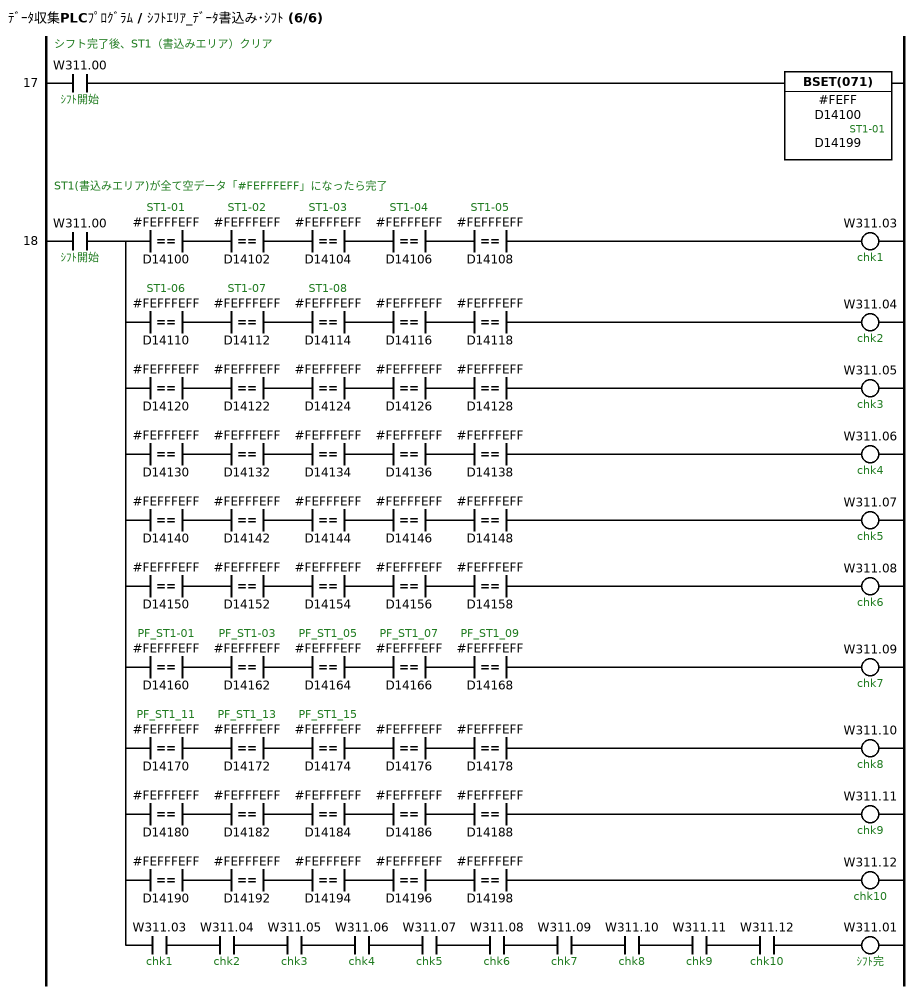
; [picture p24: ﾃﾞｰﾀ収集PLCﾌﾟﾛｸﾞﾗﾑ / ｼﾌﾄｴﾘｱ_ﾃﾞｰﾀ書込み･ｼﾌﾄ, rungs 17-18]
; rung 17: シフト完了後、ST1（書込みエリア）クリア
LD W311.00  ; ｼﾌﾄ開始
BSET(071) #FEFF D14100 D14199  ; ST1-01
; rung 18: ST1(書込みエリア)が全て空データ「#FEFFFEFF」になったら完了
LD W311.00  ; ｼﾌﾄ開始
OUT TR0
AND=L(301) #FEFFFEFF D14100  ; ST1-01
AND=L(301) #FEFFFEFF D14102  ; ST1-02
AND=L(301) #FEFFFEFF D14104  ; ST1-03
AND=L(301) #FEFFFEFF D14106  ; ST1-04
AND=L(301) #FEFFFEFF D14108  ; ST1-05
OUT W311.03  ; chk1
LD TR0
AND=L(301) #FEFFFEFF D14110  ; ST1-06
AND=L(301) #FEFFFEFF D14112  ; ST1-07
AND=L(301) #FEFFFEFF D14114  ; ST1-08
AND=L(301) #FEFFFEFF D14116
AND=L(301) #FEFFFEFF D14118
OUT W311.04  ; chk2
LD TR0
AND=L(301) #FEFFFEFF D14120
AND=L(301) #FEFFFEFF D14122
AND=L(301) #FEFFFEFF D14124
AND=L(301) #FEFFFEFF D14126
AND=L(301) #FEFFFEFF D14128
OUT W311.05  ; chk3
LD TR0
AND=L(301) #FEFFFEFF D14130
AND=L(301) #FEFFFEFF D14132
AND=L(301) #FEFFFEFF D14134
AND=L(301) #FEFFFEFF D14136
AND=L(301) #FEFFFEFF D14138
OUT W311.06  ; chk4
LD TR0
AND=L(301) #FEFFFEFF D14140
AND=L(301) #FEFFFEFF D14142
AND=L(301) #FEFFFEFF D14144
AND=L(301) #FEFFFEFF D14146
AND=L(301) #FEFFFEFF D14148
OUT W311.07  ; chk5
LD TR0
AND=L(301) #FEFFFEFF D14150
AND=L(301) #FEFFFEFF D14152
AND=L(301) #FEFFFEFF D14154
AND=L(301) #FEFFFEFF D14156
AND=L(301) #FEFFFEFF D14158
OUT W311.08  ; chk6
LD TR0
AND=L(301) #FEFFFEFF D14160  ; PF_ST1-01
AND=L(301) #FEFFFEFF D14162  ; PF_ST1-03
AND=L(301) #FEFFFEFF D14164  ; PF_ST1_05
AND=L(301) #FEFFFEFF D14166  ; PF_ST1_07
AND=L(301) #FEFFFEFF D14168  ; PF_ST1_09
OUT W311.09  ; chk7
LD TR0
AND=L(301) #FEFFFEFF D14170  ; PF_ST1_11
AND=L(301) #FEFFFEFF D14172  ; PF_ST1_13
AND=L(301) #FEFFFEFF D14174  ; PF_ST1_15
AND=L(301) #FEFFFEFF D14176
AND=L(301) #FEFFFEFF D14178
OUT W311.10  ; chk8
LD TR0
AND=L(301) #FEFFFEFF D14180
AND=L(301) #FEFFFEFF D14182
AND=L(301) #FEFFFEFF D14184
AND=L(301) #FEFFFEFF D14186
AND=L(301) #FEFFFEFF D14188
OUT W311.11  ; chk9
LD TR0
AND=L(301) #FEFFFEFF D14190
AND=L(301) #FEFFFEFF D14192
AND=L(301) #FEFFFEFF D14194
AND=L(301) #FEFFFEFF D14196
AND=L(301) #FEFFFEFF D14198
OUT W311.12  ; chk10
LD TR0
AND W311.03  ; chk1
AND W311.04  ; chk2
AND W311.05  ; chk3
AND W311.06  ; chk4
AND W311.07  ; chk5
AND W311.08  ; chk6
AND W311.09  ; chk7
AND W311.10  ; chk8
AND W311.11  ; chk9
AND W311.12  ; chk10
OUT W311.01  ; ｼﾌﾄ完

### Section ｼﾌﾄｴﾘｱ_ﾃﾞｰﾀ読出し

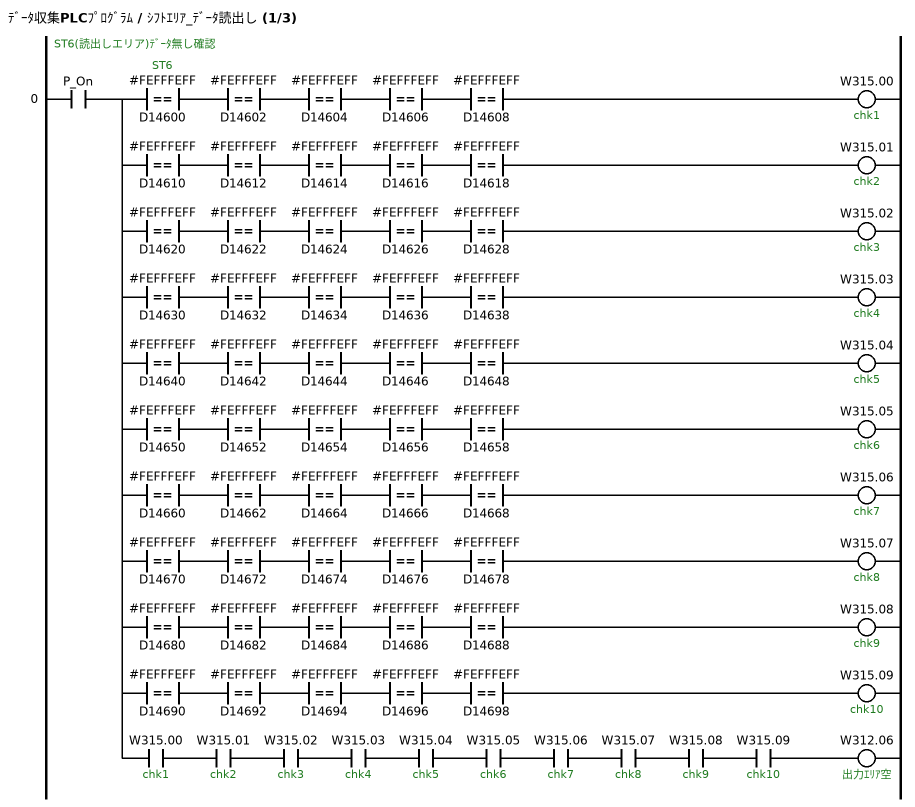
; rung 0: ST6(読出しエリア)ﾃﾞｰﾀ無し確認
LD P_On
OUT TR0
AND=L(301) #FEFFFEFF D14600  ; ST6
AND=L(301) #FEFFFEFF D14602
AND=L(301) #FEFFFEFF D14604
AND=L(301) #FEFFFEFF D14606
AND=L(301) #FEFFFEFF D14608
OUT W315.00  ; chk1
LD TR0
AND=L(301) #FEFFFEFF D14610
AND=L(301) #FEFFFEFF D14612
AND=L(301) #FEFFFEFF D14614
AND=L(301) #FEFFFEFF D14616
AND=L(301) #FEFFFEFF D14618
OUT W315.01  ; chk2
LD TR0
AND=L(301) #FEFFFEFF D14620
AND=L(301) #FEFFFEFF D14622
AND=L(301) #FEFFFEFF D14624
AND=L(301) #FEFFFEFF D14626
AND=L(301) #FEFFFEFF D14628
OUT W315.02  ; chk3
LD TR0
AND=L(301) #FEFFFEFF D14630
AND=L(301) #FEFFFEFF D14632
AND=L(301) #FEFFFEFF D14634
AND=L(301) #FEFFFEFF D14636
AND=L(301) #FEFFFEFF D14638
OUT W315.03  ; chk4
LD TR0
AND=L(301) #FEFFFEFF D14640
AND=L(301) #FEFFFEFF D14642
AND=L(301) #FEFFFEFF D14644
AND=L(301) #FEFFFEFF D14646
AND=L(301) #FEFFFEFF D14648
OUT W315.04  ; chk5
LD TR0
AND=L(301) #FEFFFEFF D14650
AND=L(301) #FEFFFEFF D14652
AND=L(301) #FEFFFEFF D14654
AND=L(301) #FEFFFEFF D14656
AND=L(301) #FEFFFEFF D14658
OUT W315.05  ; chk6
LD TR0
AND=L(301) #FEFFFEFF D14660
AND=L(301) #FEFFFEFF D14662
AND=L(301) #FEFFFEFF D14664
AND=L(301) #FEFFFEFF D14666
AND=L(301) #FEFFFEFF D14668
OUT W315.06  ; chk7
LD TR0
AND=L(301) #FEFFFEFF D14670
AND=L(301) #FEFFFEFF D14672
AND=L(301) #FEFFFEFF D14674
AND=L(301) #FEFFFEFF D14676
AND=L(301) #FEFFFEFF D14678
OUT W315.07  ; chk8
LD TR0
AND=L(301) #FEFFFEFF D14680
AND=L(301) #FEFFFEFF D14682
AND=L(301) #FEFFFEFF D14684
AND=L(301) #FEFFFEFF D14686
AND=L(301) #FEFFFEFF D14688
OUT W315.08  ; chk9
LD TR0
AND=L(301) #FEFFFEFF D14690
AND=L(301) #FEFFFEFF D14692
AND=L(301) #FEFFFEFF D14694
AND=L(301) #FEFFFEFF D14696
AND=L(301) #FEFFFEFF D14698
OUT W315.09  ; chk10
LD TR0
AND W315.00  ; chk1
AND W315.01  ; chk2
AND W315.02  ; chk3
AND W315.03  ; chk4
AND W315.04  ; chk5
AND W315.05  ; chk6
AND W315.06  ; chk7
AND W315.07  ; chk8
AND W315.08  ; chk9
AND W315.09  ; chk10
OUT W312.06  ; 出力ｴﾘｱ空

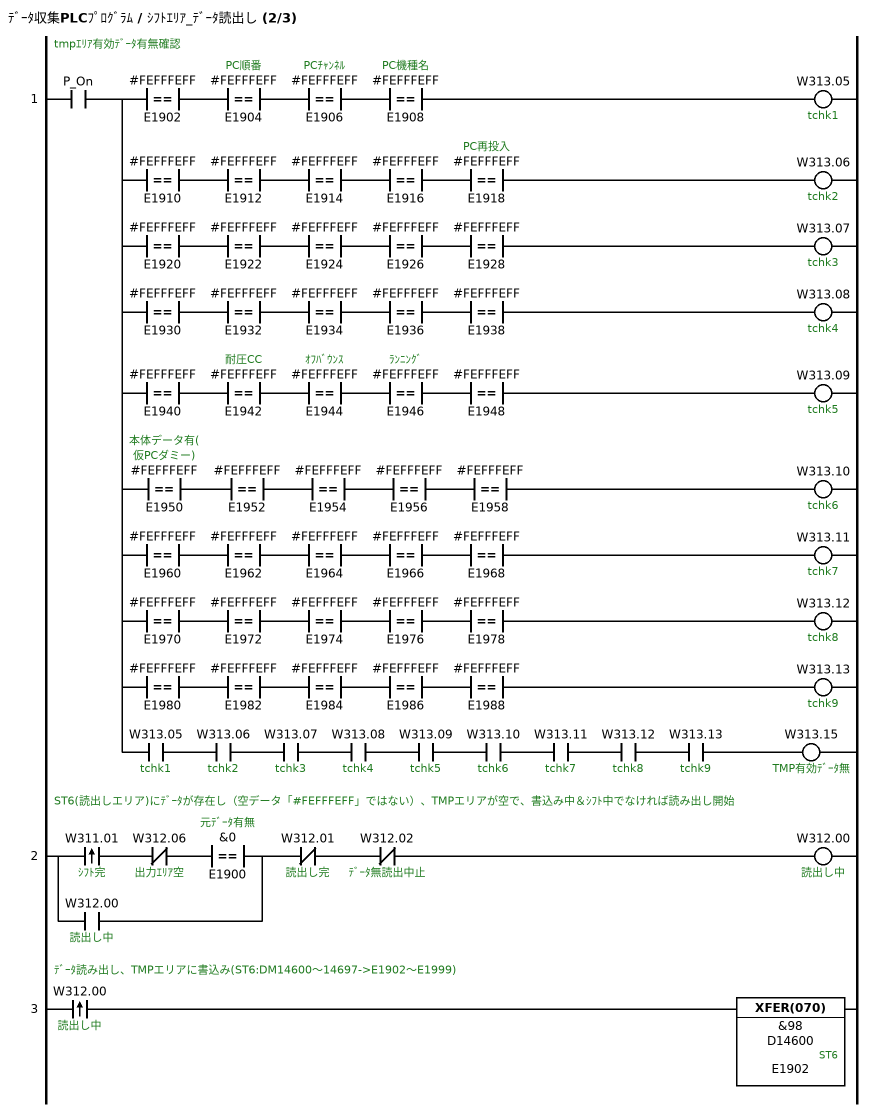
; rung 1: tmpｴﾘｱ有効ﾃﾞｰﾀ有無確認
LD P_On
OUT TR0
AND=L(301) #FEFFFEFF E1902
AND=L(301) #FEFFFEFF E1904  ; PC順番
AND=L(301) #FEFFFEFF E1906  ; PCﾁｬﾝﾈﾙ
AND=L(301) #FEFFFEFF E1908  ; PC機種名
OUT W313.05  ; tchk1
LD TR0
AND=L(301) #FEFFFEFF E1910
AND=L(301) #FEFFFEFF E1912
AND=L(301) #FEFFFEFF E1914
AND=L(301) #FEFFFEFF E1916
AND=L(301) #FEFFFEFF E1918  ; PC再投入
OUT W313.06  ; tchk2
LD TR0
AND=L(301) #FEFFFEFF E1920
AND=L(301) #FEFFFEFF E1922
AND=L(301) #FEFFFEFF E1924
AND=L(301) #FEFFFEFF E1926
AND=L(301) #FEFFFEFF E1928
OUT W313.07  ; tchk3
LD TR0
AND=L(301) #FEFFFEFF E1930
AND=L(301) #FEFFFEFF E1932
AND=L(301) #FEFFFEFF E1934
AND=L(301) #FEFFFEFF E1936
AND=L(301) #FEFFFEFF E1938
OUT W313.08  ; tchk4
LD TR0
AND=L(301) #FEFFFEFF E1940
AND=L(301) #FEFFFEFF E1942  ; 耐圧CC
AND=L(301) #FEFFFEFF E1944  ; ｵﾌﾊﾞｳﾝｽ
AND=L(301) #FEFFFEFF E1946  ; ﾗﾝﾆﾝｸﾞ
AND=L(301) #FEFFFEFF E1948
OUT W313.09  ; tchk5
LD TR0
AND=L(301) #FEFFFEFF E1950  ; 本体データ有(仮PCダミー)
AND=L(301) #FEFFFEFF E1952
AND=L(301) #FEFFFEFF E1954
AND=L(301) #FEFFFEFF E1956
AND=L(301) #FEFFFEFF E1958
OUT W313.10  ; tchk6
LD TR0
AND=L(301) #FEFFFEFF E1960
AND=L(301) #FEFFFEFF E1962
AND=L(301) #FEFFFEFF E1964
AND=L(301) #FEFFFEFF E1966
AND=L(301) #FEFFFEFF E1968
OUT W313.11  ; tchk7
LD TR0
AND=L(301) #FEFFFEFF E1970
AND=L(301) #FEFFFEFF E1972
AND=L(301) #FEFFFEFF E1974
AND=L(301) #FEFFFEFF E1976
AND=L(301) #FEFFFEFF E1978
OUT W313.12  ; tchk8
LD TR0
AND=L(301) #FEFFFEFF E1980
AND=L(301) #FEFFFEFF E1982
AND=L(301) #FEFFFEFF E1984
AND=L(301) #FEFFFEFF E1986
AND=L(301) #FEFFFEFF E1988
OUT W313.13  ; tchk9
LD TR0
AND W313.05  ; tchk1
AND W313.06  ; tchk2
AND W313.07  ; tchk3
AND W313.08  ; tchk4
AND W313.09  ; tchk5
AND W313.10  ; tchk6
AND W313.11  ; tchk7
AND W313.12  ; tchk8
AND W313.13  ; tchk9
OUT W313.15  ; TMP有効ﾃﾞｰﾀ無
; rung 2: ST6(読出しエリア)にﾃﾞｰﾀが存在し（空データ「#FEFFFEFF」ではない）、TMPエリアが空で、書込み中＆ｼﾌﾄ中でなければ読み出し開始
@LD W311.01  ; ｼﾌﾄ完
ANDNOT W312.06  ; 出力ｴﾘｱ空
AND=(300) &0 E1900  ; 元ﾃﾞｰﾀ有無
OR W312.00  ; 読出し中
ANDNOT W312.01  ; 読出し完
ANDNOT W312.02  ; ﾃﾞｰﾀ無読出中止
OUT W312.00  ; 読出し中
; rung 3: ﾃﾞｰﾀ読み出し、TMPエリアに書込み(ST6:DM14600～14697->E1902～E1999)
@LD W312.00  ; 読出し中
XFER(070) &98 D14600 E1902  ; ST6

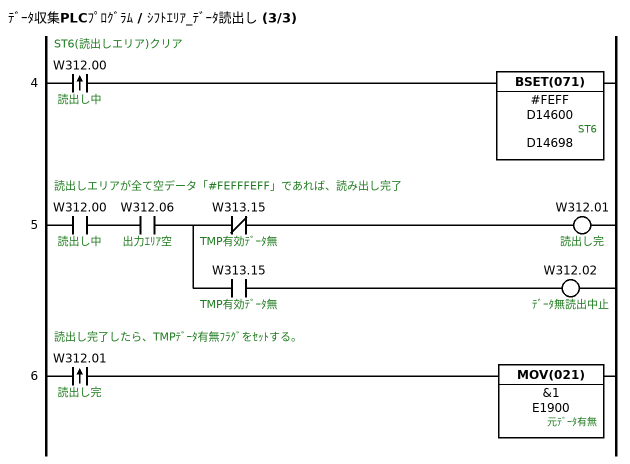
; rung 4: ST6(読出しエリア)クリア
@LD W312.00  ; 読出し中
BSET(071) #FEFF D14600 D14698  ; ST6
; rung 5: 読出しエリアが全て空データ「#FEFFFEFF」であれば、読み出し完了
LD W312.00  ; 読出し中
AND W312.06  ; 出力ｴﾘｱ空
OUT TR0
ANDNOT W313.15  ; TMP有効ﾃﾞｰﾀ無
OUT W312.01  ; 読出し完
LD TR0
AND W313.15  ; TMP有効ﾃﾞｰﾀ無
OUT W312.02  ; ﾃﾞｰﾀ無読出中止
; rung 6: 読出し完了したら、TMPﾃﾞｰﾀ有無ﾌﾗｸﾞをｾｯﾄする。
@LD W312.01  ; 読出し完
MOV(021) &1 E1900  ; 元ﾃﾞｰﾀ有無

### Section ｼﾌﾄｴﾘｱ_ﾃﾞｰﾀｸﾘｱ

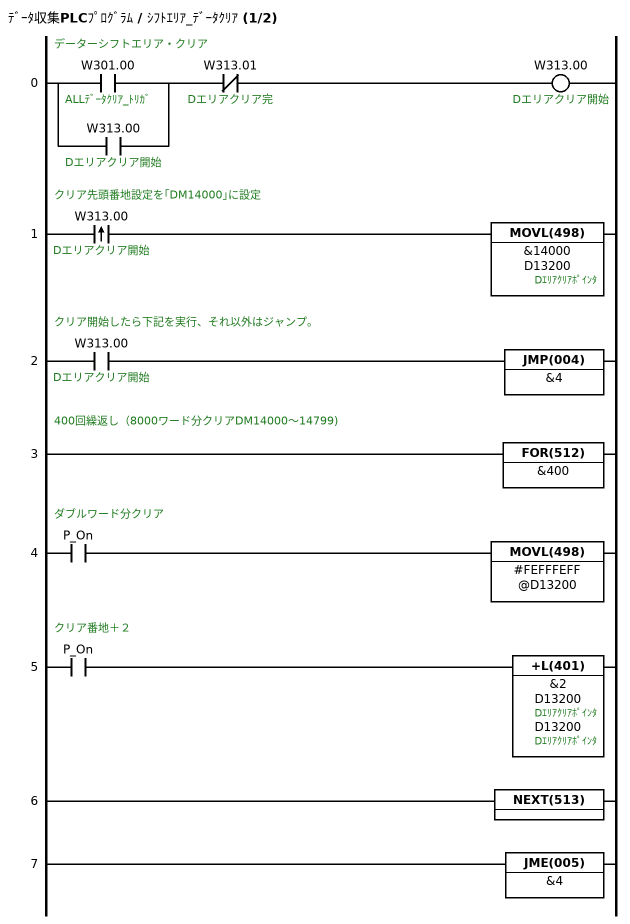
; rung 0: データーシフトエリア・クリア
LD W301.00  ; ALLﾃﾞｰﾀｸﾘｱ_ﾄﾘｶﾞ
OR W313.00  ; Dエリアクリア開始
ANDNOT W313.01  ; Dエリアクリア完
OUT W313.00  ; Dエリアクリア開始
; rung 1: クリア先頭番地設定を｢DM14000｣に設定
@LD W313.00  ; Dエリアクリア開始
MOVL(498) &14000 D13200  ; Dｴﾘｱｸﾘｱﾎﾟｲﾝﾀ
; rung 2: クリア開始したら下記を実行、それ以外はジャンプ。
LD W313.00  ; Dエリアクリア開始
JMP(004) &4
; rung 3: 400回繰返し（8000ワード分クリアDM14000～14799)
FOR(512) &400
; rung 4: ダブルワード分クリア
LD P_On
MOVL(498) #FEFFFEFF @D13200
; rung 5: クリア番地＋２
LD P_On
+L(401) &2 D13200 D13200  ; Dｴﾘｱｸﾘｱﾎﾟｲﾝﾀ
; rung 6
NEXT(513)
; rung 7
JME(005) &4

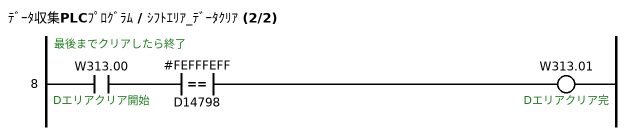
; rung 8: 最後までクリアしたら終了
LD W313.00  ; Dエリアクリア開始
AND=L(301) #FEFFFEFF D14798
OUT W313.01  ; Dエリアクリア完

### Section ｽﾀｯｸｴﾘｱ_ﾃﾞｰﾀ書込み

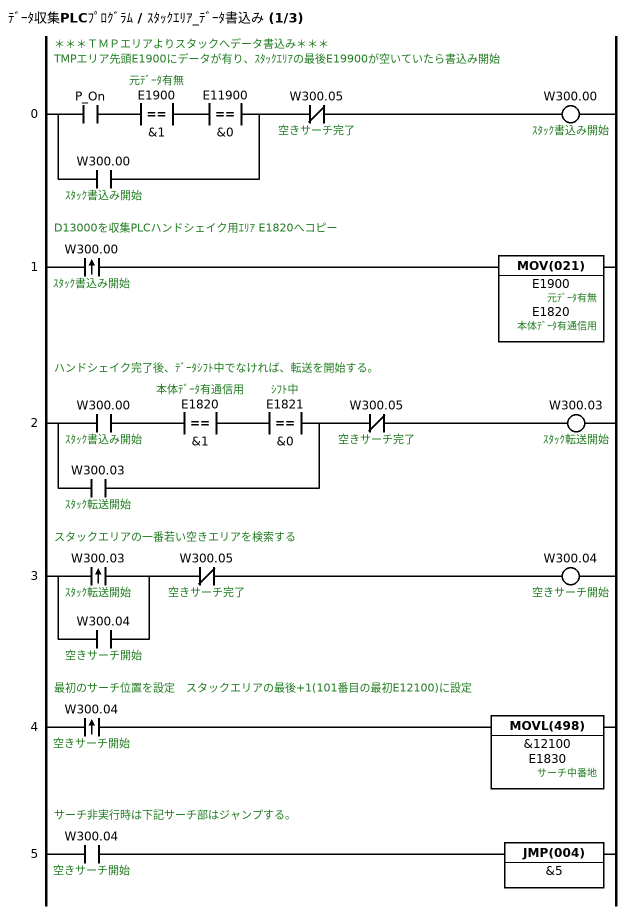
; rung 0: ＊＊＊ＴＭＰエリアよりスタックへデータ書込み＊＊＊ / TMPエリア先頭E1900にデータが有り、ｽﾀｯｸｴﾘｱの最後E19900が空いていたら書込み開始
LD P_On
AND=(300) E1900 &1  ; 元ﾃﾞｰﾀ有無
AND=(300) E11900 &0
OR W300.00  ; ｽﾀｯｸ書込み開始
ANDNOT W300.05  ; 空きサーチ完了
OUT W300.00  ; ｽﾀｯｸ書込み開始
; rung 1: D13000を収集PLCハンドシェイク用ｴﾘｱ E1820へコピー
@LD W300.00  ; ｽﾀｯｸ書込み開始
MOV(021) E1900 E1820  ; 元ﾃﾞｰﾀ有無, 本体ﾃﾞｰﾀ有通信用
; rung 2: ハンドシェイク完了後、ﾃﾞｰﾀｼﾌﾄ中でなければ、転送を開始する。
LD W300.00  ; ｽﾀｯｸ書込み開始
AND=(300) E1820 &1  ; 本体ﾃﾞｰﾀ有通信用
AND=(300) E1821 &0  ; ｼﾌﾄ中
OR W300.03  ; ｽﾀｯｸ転送開始
ANDNOT W300.05  ; 空きサーチ完了
OUT W300.03  ; ｽﾀｯｸ転送開始
; rung 3: スタックエリアの一番若い空きエリアを検索する
@LD W300.03  ; ｽﾀｯｸ転送開始
OR W300.04  ; 空きサーチ開始
ANDNOT W300.05  ; 空きサーチ完了
OUT W300.04  ; 空きサーチ開始
; rung 4: 最初のサーチ位置を設定　スタックエリアの最後+1(101番目の最初E12100)に設定
@LD W300.04  ; 空きサーチ開始
MOVL(498) &12100 E1830  ; サーチ中番地
; rung 5: サーチ非実行時は下記サーチ部はジャンプする。
LD W300.04  ; 空きサーチ開始
JMP(004) &5

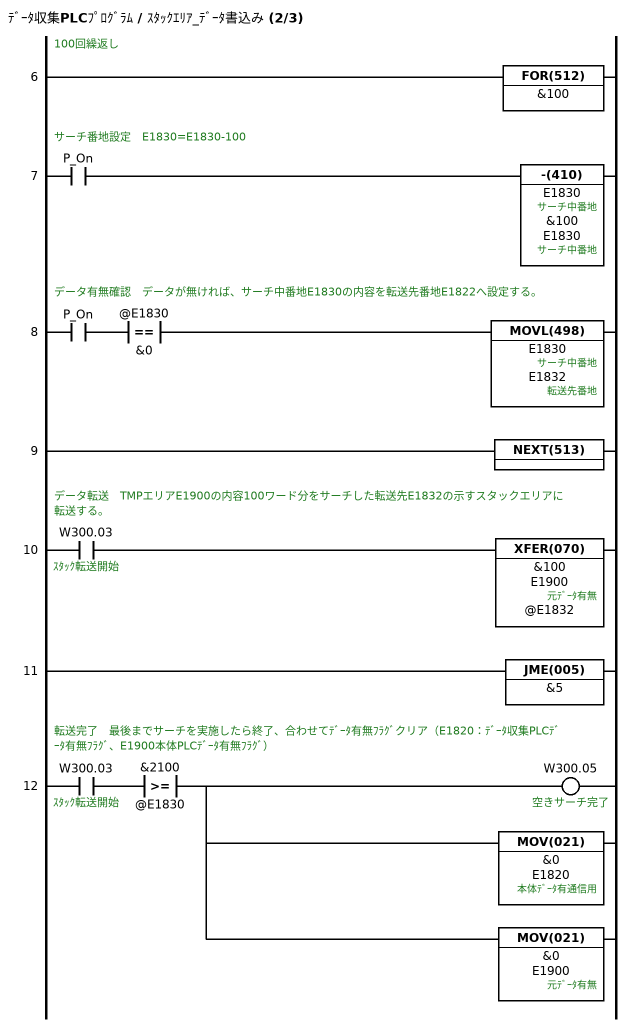
; rung 6: 100回繰返し
FOR(512) &100
; rung 7: サーチ番地設定　E1830=E1830-100
LD P_On
-(410) E1830 &100 E1830  ; サーチ中番地
; rung 8: データ有無確認　データが無ければ、サーチ中番地E1830の内容を転送先番地E1822へ設定する。
LD P_On
AND=(300) @E1830 &0
MOVL(498) E1830 E1832  ; サーチ中番地, 転送先番地
; rung 9
NEXT(513)
; rung 10: データ転送　TMPエリアE1900の内容100ワード分をサーチした転送先E1832の示すスタックエリアに転送する。
LD W300.03  ; ｽﾀｯｸ転送開始
XFER(070) &100 E1900 @E1832  ; 元ﾃﾞｰﾀ有無
; rung 11
JME(005) &5
; rung 12: 転送完了　最後までサーチを実施したら終了、合わせてﾃﾞｰﾀ有無ﾌﾗｸﾞクリア（E1820：ﾃﾞｰﾀ収集PLCﾃﾞｰﾀ有無ﾌﾗｸﾞ、E1900本体PLCﾃﾞｰﾀ有無ﾌﾗｸﾞ）
LD W300.03  ; ｽﾀｯｸ転送開始
AND>=(325) &2100 @E1830
OUT W300.05  ; 空きサーチ完了
MOV(021) &0 E1820  ; 本体ﾃﾞｰﾀ有通信用
MOV(021) &0 E1900  ; 元ﾃﾞｰﾀ有無

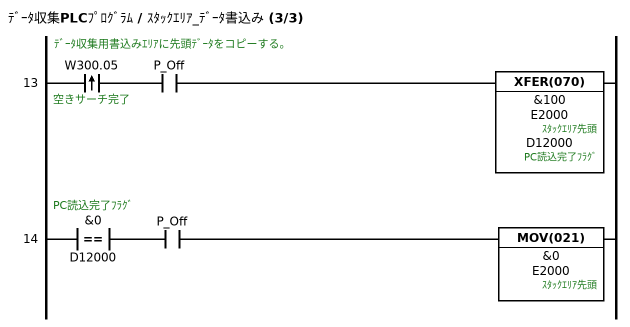
; rung 13: ﾃﾞｰﾀ収集用書込みｴﾘｱに先頭ﾃﾞｰﾀをコピーする。
@LD W300.05  ; 空きサーチ完了
AND P_Off
XFER(070) &100 E2000 D12000  ; ｽﾀｯｸｴﾘｱ先頭, PC読込完了ﾌﾗｸﾞ
; rung 14
LD=(300) &0 D12000  ; PC読込完了ﾌﾗｸﾞ
AND P_Off
MOV(021) &0 E2000  ; ｽﾀｯｸｴﾘｱ先頭

### Section ｽﾀｯｸｴﾘｱ_ﾃﾞｰﾀｼﾌﾄ

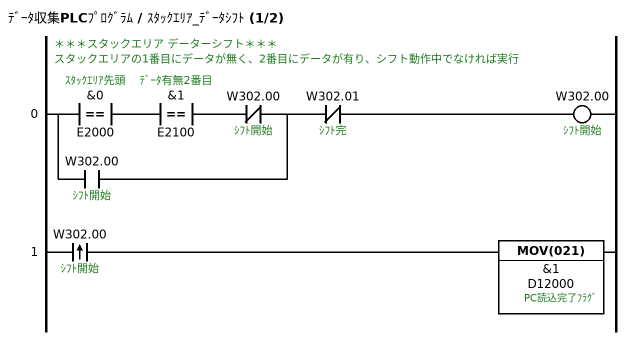
; rung 0: ＊＊＊スタックエリア データーシフト＊＊＊ / スタックエリアの1番目にデータが無く、2番目にデータが有り、シフト動作中でなければ実行
LD=(300) &0 E2000  ; ｽﾀｯｸｴﾘｱ先頭
AND=(300) &1 E2100  ; ﾃﾞｰﾀ有無2番目
ANDNOT W302.00  ; ｼﾌﾄ開始
OR W302.00  ; ｼﾌﾄ開始
ANDNOT W302.01  ; ｼﾌﾄ完
OUT W302.00  ; ｼﾌﾄ開始
; rung 1
@LD W302.00  ; ｼﾌﾄ開始
MOV(021) &1 D12000  ; PC読込完了ﾌﾗｸﾞ

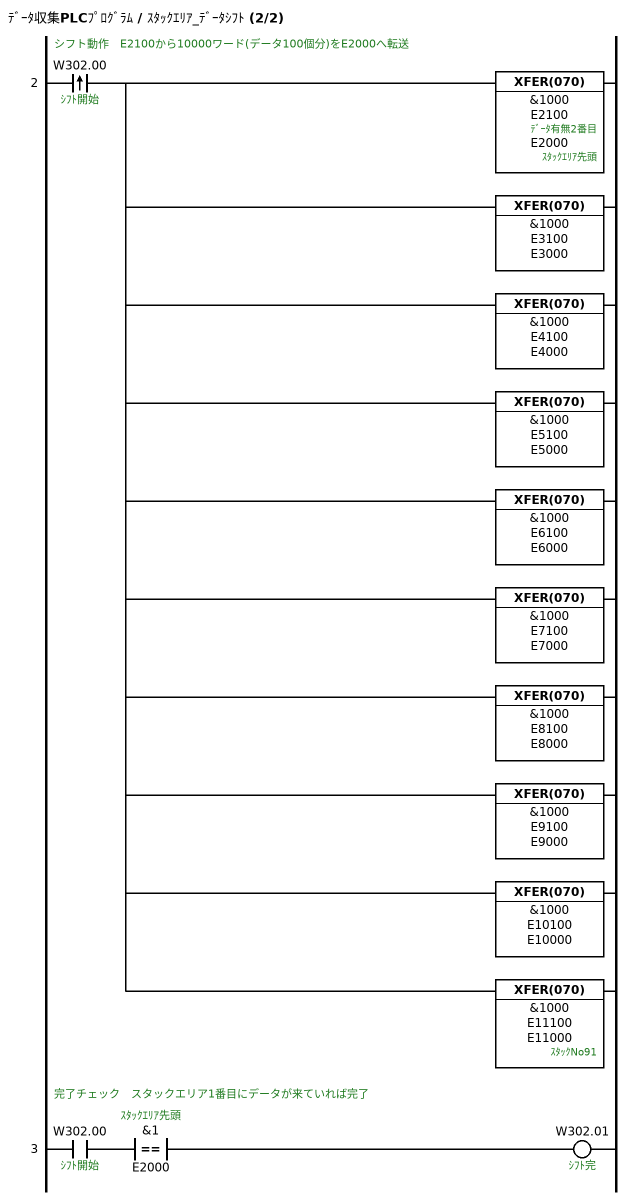
; rung 2: シフト動作　E2100から10000ワード(データ100個分)をE2000へ転送
@LD W302.00  ; ｼﾌﾄ開始
XFER(070) &1000 E2100 E2000  ; ﾃﾞｰﾀ有無2番目, ｽﾀｯｸｴﾘｱ先頭
XFER(070) &1000 E3100 E3000
XFER(070) &1000 E4100 E4000
XFER(070) &1000 E5100 E5000
XFER(070) &1000 E6100 E6000
XFER(070) &1000 E7100 E7000
XFER(070) &1000 E8100 E8000
XFER(070) &1000 E9100 E9000
XFER(070) &1000 E10100 E10000
XFER(070) &1000 E11100 E11000  ; ｽﾀｯｸNo91
; rung 3: 完了チェック　スタックエリア1番目にデータが来ていれば完了
LD W302.00  ; ｼﾌﾄ開始
AND=(300) &1 E2000  ; ｽﾀｯｸｴﾘｱ先頭
OUT W302.01  ; ｼﾌﾄ完

### Section ｽﾀｯｸｴﾘｱ_ﾃﾞｰﾀｸﾘｱ

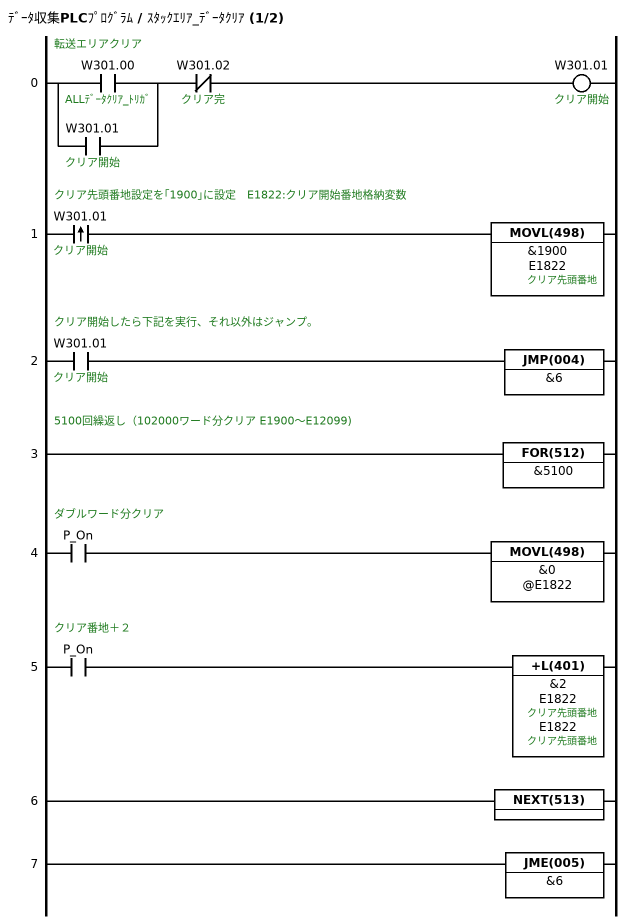
; rung 0: 転送エリアクリア
LD W301.00  ; ALLﾃﾞｰﾀｸﾘｱ_ﾄﾘｶﾞ
OR W301.01  ; クリア開始
ANDNOT W301.02  ; クリア完
OUT W301.01  ; クリア開始
; rung 1: クリア先頭番地設定を｢1900｣に設定　E1822:クリア開始番地格納変数
@LD W301.01  ; クリア開始
MOVL(498) &1900 E1822  ; クリア先頭番地
; rung 2: クリア開始したら下記を実行、それ以外はジャンプ。
LD W301.01  ; クリア開始
JMP(004) &6
; rung 3: 5100回繰返し（102000ワード分クリア E1900～E12099)
FOR(512) &5100
; rung 4: ダブルワード分クリア
LD P_On
MOVL(498) &0 @E1822
; rung 5: クリア番地＋２
LD P_On
+L(401) &2 E1822 E1822  ; クリア先頭番地
; rung 6
NEXT(513)
; rung 7
JME(005) &6

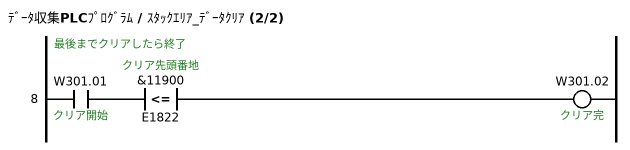
; rung 8: 最後までクリアしたら終了
LD W301.01  ; クリア開始
AND<=(315) &11900 E1822  ; クリア先頭番地
OUT W301.02  ; クリア完

### Section PCﾃﾞｰﾀ吸上げﾊﾝﾄﾞｼｪｲｸ

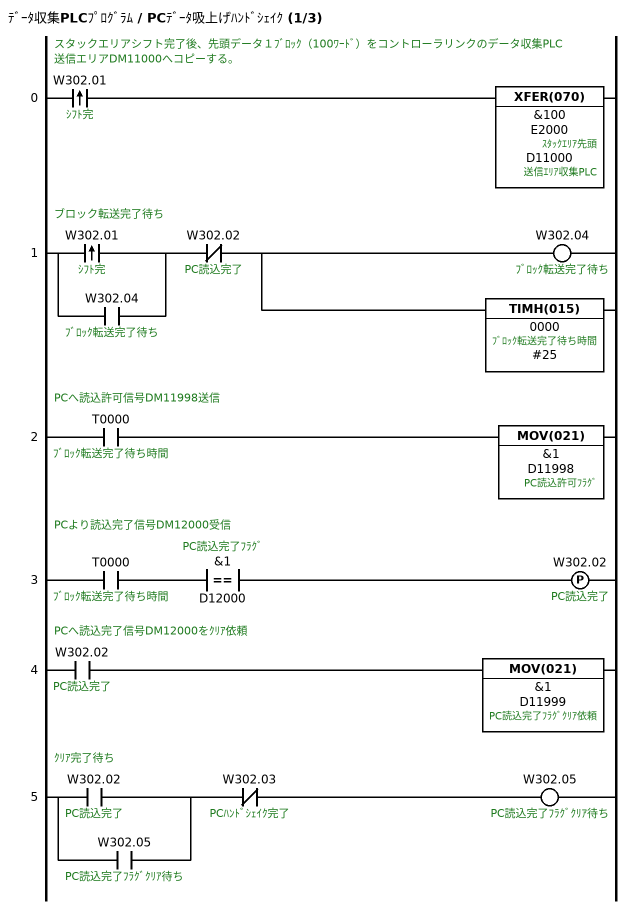
; rung 0: スタックエリアシフト完了後、先頭データ１ﾌﾞﾛｯｸ（100ﾜｰﾄﾞ）をコントローラリンクのデータ収集PLC送信エリアDM11000へコピーする。
@LD W302.01  ; ｼﾌﾄ完
XFER(070) &100 E2000 D11000  ; ｽﾀｯｸｴﾘｱ先頭, 送信ｴﾘｱ収集PLC
; rung 1: ブロック転送完了待ち
@LD W302.01  ; ｼﾌﾄ完
OR W302.04  ; ﾌﾞﾛｯｸ転送完了待ち
ANDNOT W302.02  ; PC読込完了
OUT W302.04  ; ﾌﾞﾛｯｸ転送完了待ち
TIMH(015) 0000 #25  ; ﾌﾞﾛｯｸ転送完了待ち時間
; rung 2: PCへ読込許可信号DM11998送信
LD T0000  ; ﾌﾞﾛｯｸ転送完了待ち時間
MOV(021) &1 D11998  ; PC読込許可ﾌﾗｸﾞ
; rung 3: PCより読込完了信号DM12000受信
LD T0000  ; ﾌﾞﾛｯｸ転送完了待ち時間
AND=(300) &1 D12000  ; PC読込完了ﾌﾗｸﾞ
DIFU(013) W302.02  ; PC読込完了
; rung 4: PCへ読込完了信号DM12000をｸﾘｱ依頼
LD W302.02  ; PC読込完了
MOV(021) &1 D11999  ; PC読込完了ﾌﾗｸﾞｸﾘｱ依頼
; rung 5: ｸﾘｱ完了待ち
LD W302.02  ; PC読込完了
OR W302.05  ; PC読込完了ﾌﾗｸﾞｸﾘｱ待ち
ANDNOT W302.03  ; PCﾊﾝﾄﾞｼｪｲｸ完了
OUT W302.05  ; PC読込完了ﾌﾗｸﾞｸﾘｱ待ち

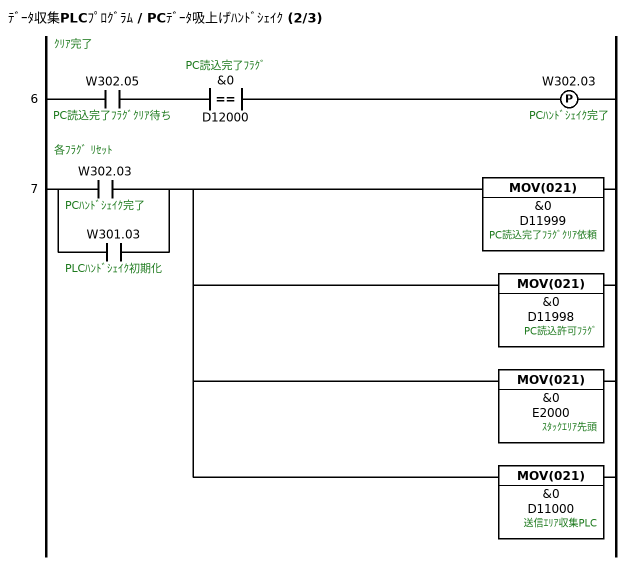
; rung 6: ｸﾘｱ完了
LD W302.05  ; PC読込完了ﾌﾗｸﾞｸﾘｱ待ち
AND=(300) &0 D12000  ; PC読込完了ﾌﾗｸﾞ
DIFU(013) W302.03  ; PCﾊﾝﾄﾞｼｪｲｸ完了
; rung 7: 各ﾌﾗｸﾞ ﾘｾｯﾄ
LD W302.03  ; PCﾊﾝﾄﾞｼｪｲｸ完了
OR W301.03  ; PLCﾊﾝﾄﾞｼｪｲｸ初期化
MOV(021) &0 D11999  ; PC読込完了ﾌﾗｸﾞｸﾘｱ依頼
MOV(021) &0 D11998  ; PC読込許可ﾌﾗｸﾞ
MOV(021) &0 E2000  ; ｽﾀｯｸｴﾘｱ先頭
MOV(021) &0 D11000  ; 送信ｴﾘｱ収集PLC

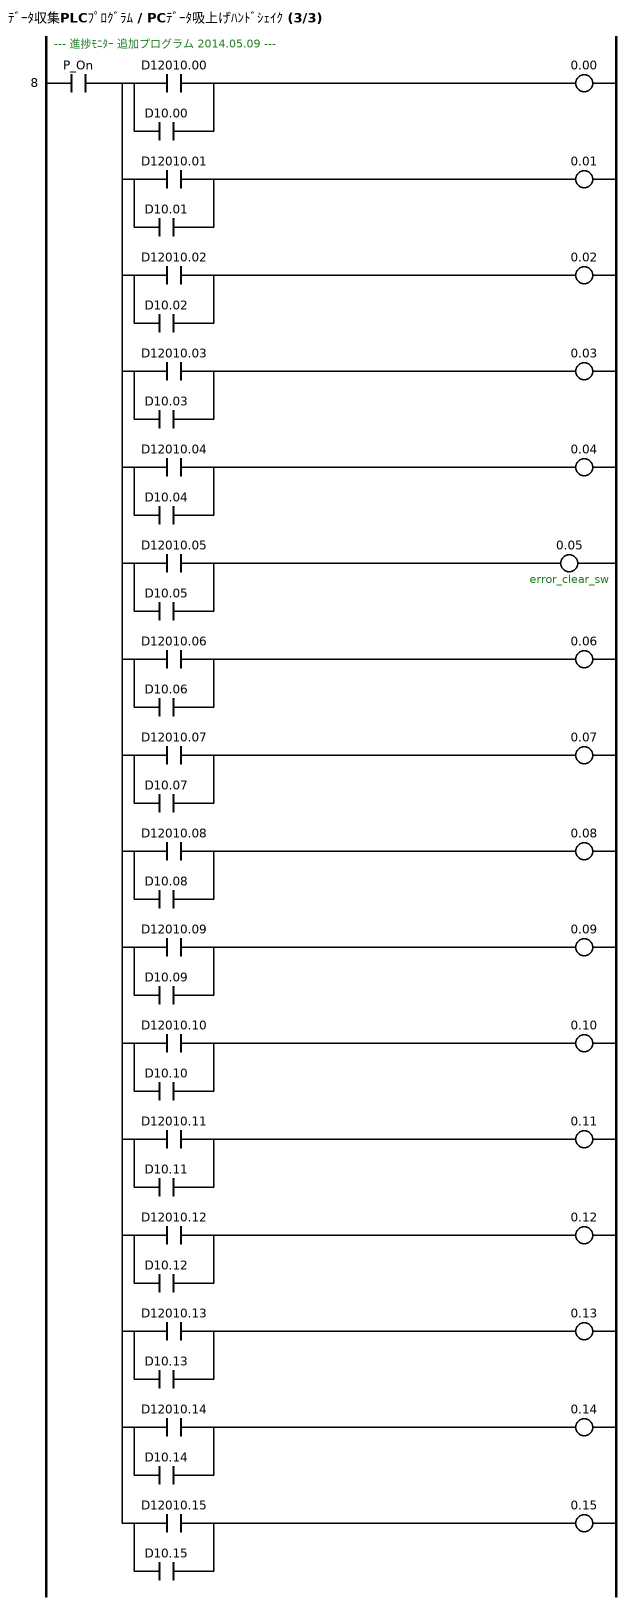
; rung 8: --- 進捗ﾓﾆﾀｰ 追加プログラム 2014.05.09 ---
LD P_On
OUT TR0
LD D12010.00
OR D10.00
ANDLD
OUT 0.00
LD TR0
LD D12010.01
OR D10.01
ANDLD
OUT 0.01
LD TR0
LD D12010.02
OR D10.02
ANDLD
OUT 0.02
LD TR0
LD D12010.03
OR D10.03
ANDLD
OUT 0.03
LD TR0
LD D12010.04
OR D10.04
ANDLD
OUT 0.04
LD TR0
LD D12010.05
OR D10.05
ANDLD
OUT 0.05  ; error_clear_sw
LD TR0
LD D12010.06
OR D10.06
ANDLD
OUT 0.06
LD TR0
LD D12010.07
OR D10.07
ANDLD
OUT 0.07
LD TR0
LD D12010.08
OR D10.08
ANDLD
OUT 0.08
LD TR0
LD D12010.09
OR D10.09
ANDLD
OUT 0.09
LD TR0
LD D12010.10
OR D10.10
ANDLD
OUT 0.10
LD TR0
LD D12010.11
OR D10.11
ANDLD
OUT 0.11
LD TR0
LD D12010.12
OR D10.12
ANDLD
OUT 0.12
LD TR0
LD D12010.13
OR D10.13
ANDLD
OUT 0.13
LD TR0
LD D12010.14
OR D10.14
ANDLD
OUT 0.14
LD TR0
LD D12010.15
OR D10.15
ANDLD
OUT 0.15

### Section ﾃﾞﾊﾞｯｸﾞﾓﾆﾀ測定値

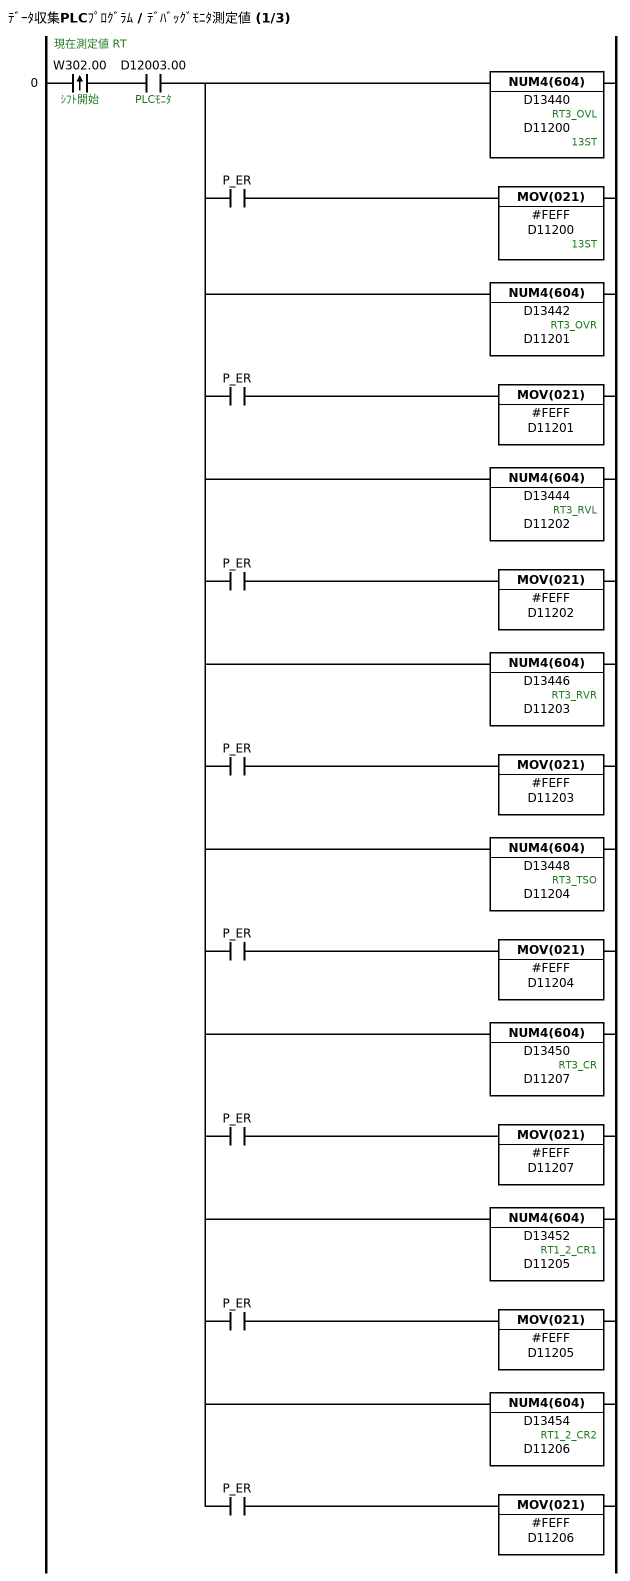
; rung 0: 現在測定値 RT
@LD W302.00  ; ｼﾌﾄ開始
AND D12003.00  ; PLCﾓﾆﾀ
OUT TR0
NUM4(604) D13440 D11200  ; RT3_OVL, 13ST
AND P_ER
MOV(021) #FEFF D11200  ; 13ST
LD TR0
NUM4(604) D13442 D11201  ; RT3_OVR
AND P_ER
MOV(021) #FEFF D11201
LD TR0
NUM4(604) D13444 D11202  ; RT3_RVL
AND P_ER
MOV(021) #FEFF D11202
LD TR0
NUM4(604) D13446 D11203  ; RT3_RVR
AND P_ER
MOV(021) #FEFF D11203
LD TR0
NUM4(604) D13448 D11204  ; RT3_TSO
AND P_ER
MOV(021) #FEFF D11204
LD TR0
NUM4(604) D13450 D11207  ; RT3_CR
AND P_ER
MOV(021) #FEFF D11207
LD TR0
NUM4(604) D13452 D11205  ; RT1_2_CR1
AND P_ER
MOV(021) #FEFF D11205
LD TR0
NUM4(604) D13454 D11206  ; RT1_2_CR2
AND P_ER
MOV(021) #FEFF D11206

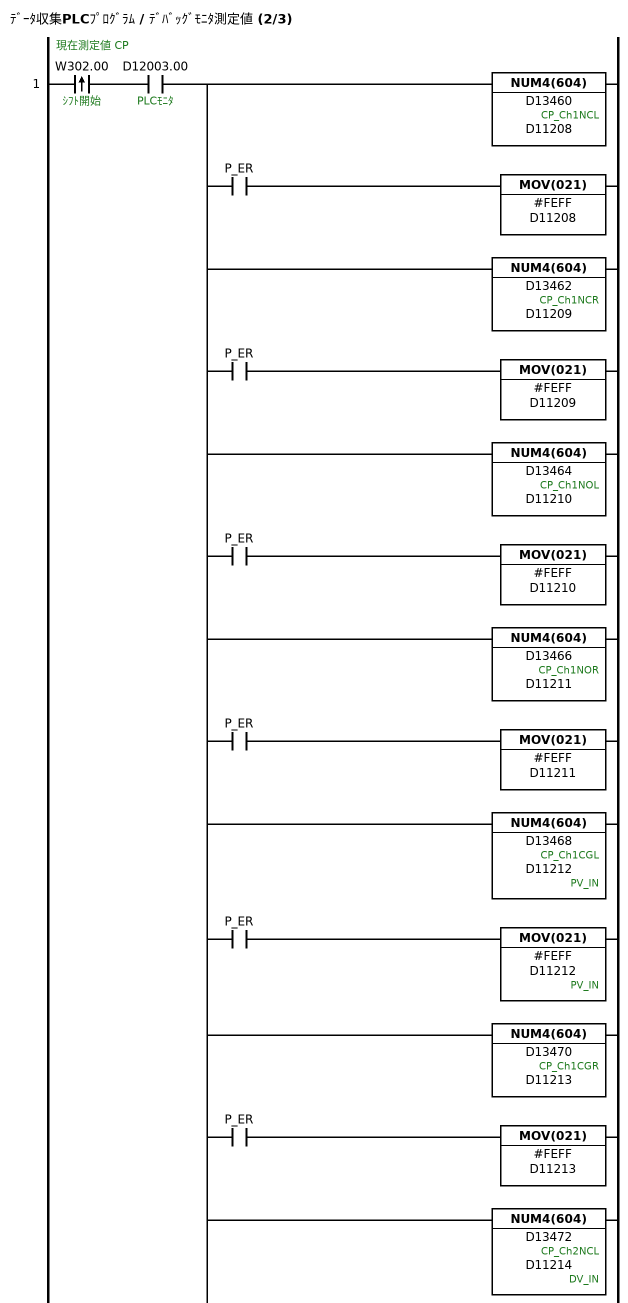

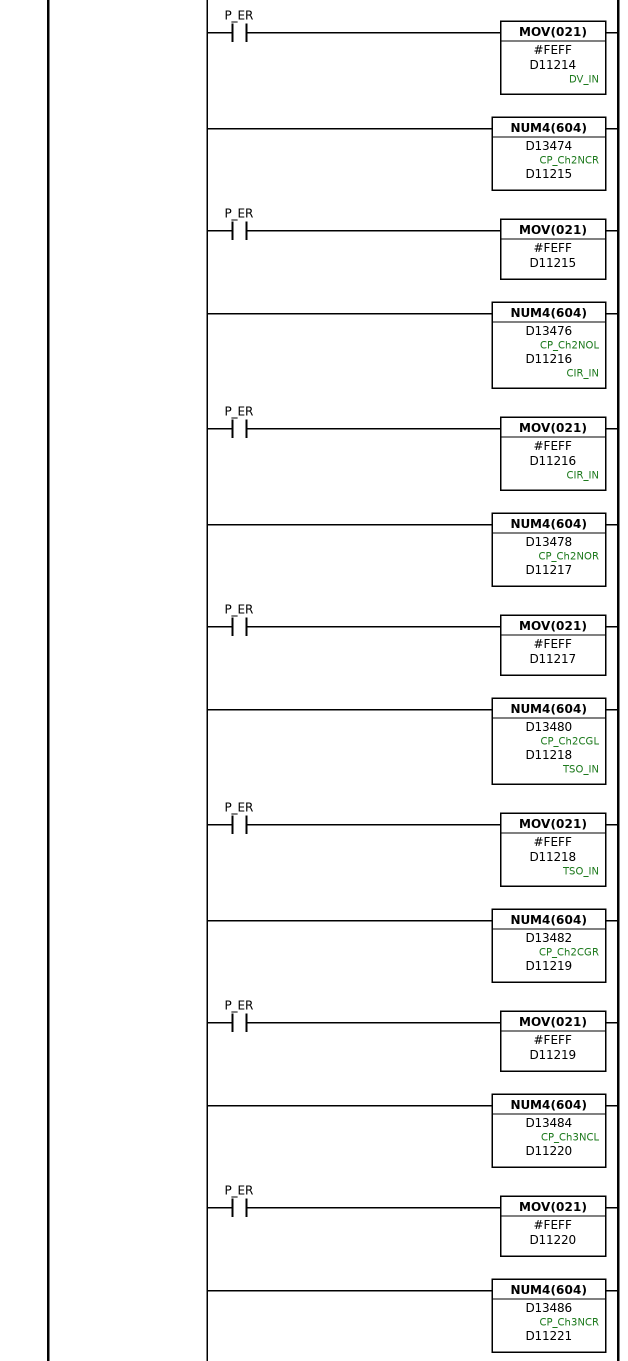

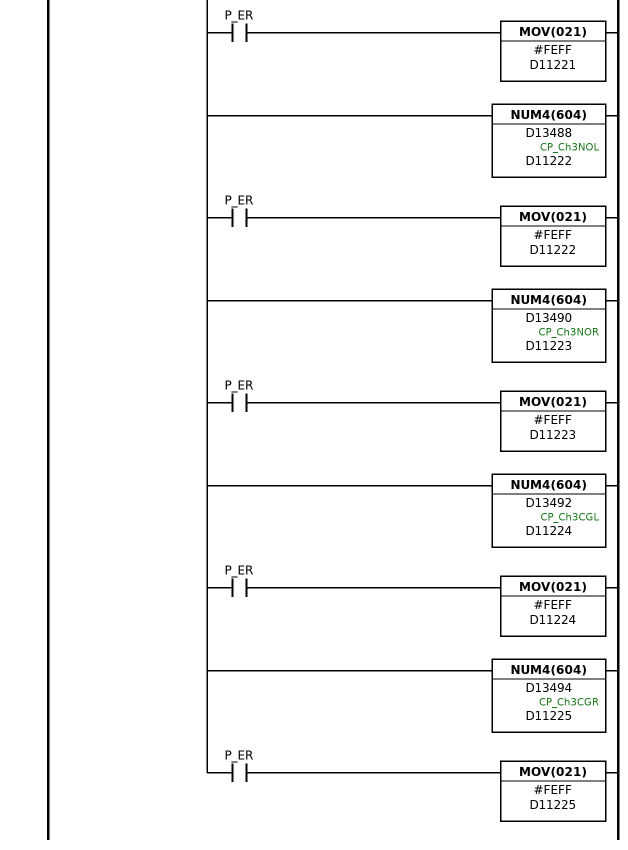
; rung 1: 現在測定値 CP
@LD W302.00  ; ｼﾌﾄ開始
AND D12003.00  ; PLCﾓﾆﾀ
OUT TR0
NUM4(604) D13460 D11208  ; CP_Ch1NCL
AND P_ER
MOV(021) #FEFF D11208
LD TR0
NUM4(604) D13462 D11209  ; CP_Ch1NCR
AND P_ER
MOV(021) #FEFF D11209
LD TR0
NUM4(604) D13464 D11210  ; CP_Ch1NOL
AND P_ER
MOV(021) #FEFF D11210
LD TR0
NUM4(604) D13466 D11211  ; CP_Ch1NOR
AND P_ER
MOV(021) #FEFF D11211
LD TR0
NUM4(604) D13468 D11212  ; CP_Ch1CGL, PV_IN
AND P_ER
MOV(021) #FEFF D11212  ; PV_IN
LD TR0
NUM4(604) D13470 D11213  ; CP_Ch1CGR
AND P_ER
MOV(021) #FEFF D11213
LD TR0
NUM4(604) D13472 D11214  ; CP_Ch2NCL, DV_IN
AND P_ER
MOV(021) #FEFF D11214  ; DV_IN
LD TR0
NUM4(604) D13474 D11215  ; CP_Ch2NCR
AND P_ER
MOV(021) #FEFF D11215
LD TR0
NUM4(604) D13476 D11216  ; CP_Ch2NOL, CIR_IN
AND P_ER
MOV(021) #FEFF D11216  ; CIR_IN
LD TR0
NUM4(604) D13478 D11217  ; CP_Ch2NOR
AND P_ER
MOV(021) #FEFF D11217
LD TR0
NUM4(604) D13480 D11218  ; CP_Ch2CGL, TSO_IN
AND P_ER
MOV(021) #FEFF D11218  ; TSO_IN
LD TR0
NUM4(604) D13482 D11219  ; CP_Ch2CGR
AND P_ER
MOV(021) #FEFF D11219
LD TR0
NUM4(604) D13484 D11220  ; CP_Ch3NCL
AND P_ER
MOV(021) #FEFF D11220
LD TR0
NUM4(604) D13486 D11221  ; CP_Ch3NCR
AND P_ER
MOV(021) #FEFF D11221
LD TR0
NUM4(604) D13488 D11222  ; CP_Ch3NOL
AND P_ER
MOV(021) #FEFF D11222
LD TR0
NUM4(604) D13490 D11223  ; CP_Ch3NOR
AND P_ER
MOV(021) #FEFF D11223
LD TR0
NUM4(604) D13492 D11224  ; CP_Ch3CGL
AND P_ER
MOV(021) #FEFF D11224
LD TR0
NUM4(604) D13494 D11225  ; CP_Ch3CGR
AND P_ER
MOV(021) #FEFF D11225

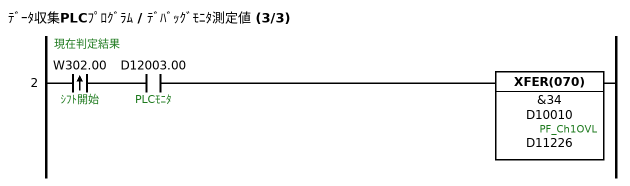
; rung 2: 現在判定結果
@LD W302.00  ; ｼﾌﾄ開始
AND D12003.00  ; PLCﾓﾆﾀ
XFER(070) &34 D10010 D11226  ; PF_Ch1OVL

### Section ﾃﾞﾊﾞｯｸﾞﾓﾆﾀSTエリア

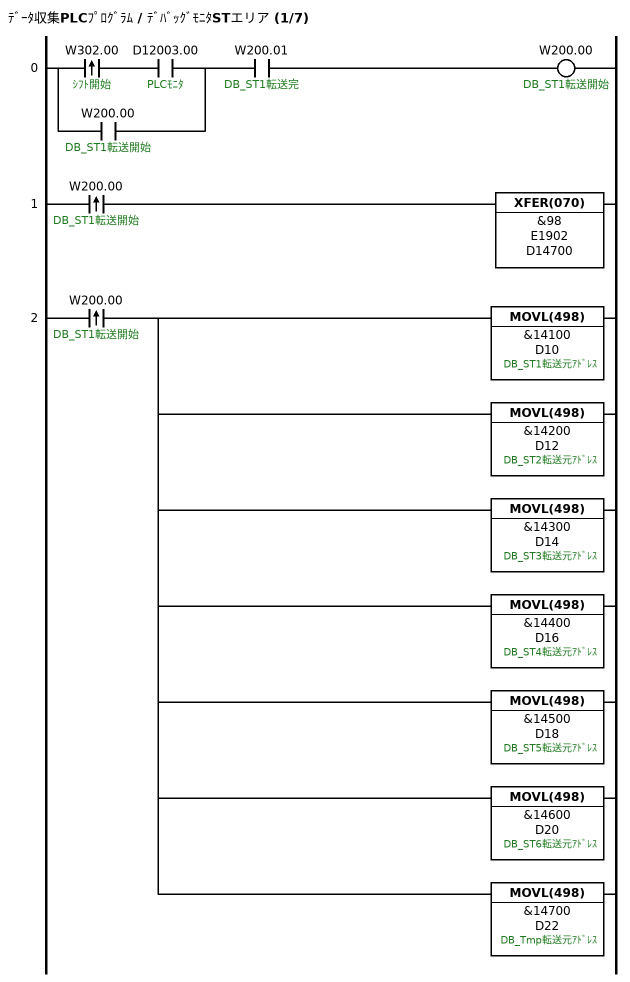
; rung 0
@LD W302.00  ; ｼﾌﾄ開始
AND D12003.00  ; PLCﾓﾆﾀ
OR W200.00  ; DB_ST1転送開始
AND W200.01  ; DB_ST1転送完
OUT W200.00  ; DB_ST1転送開始
; rung 1
@LD W200.00  ; DB_ST1転送開始
XFER(070) &98 E1902 D14700
; rung 2
@LD W200.00  ; DB_ST1転送開始
MOVL(498) &14100 D10  ; DB_ST1転送元ｱﾄﾞﾚｽ
MOVL(498) &14200 D12  ; DB_ST2転送元ｱﾄﾞﾚｽ
MOVL(498) &14300 D14  ; DB_ST3転送元ｱﾄﾞﾚｽ
MOVL(498) &14400 D16  ; DB_ST4転送元ｱﾄﾞﾚｽ
MOVL(498) &14500 D18  ; DB_ST5転送元ｱﾄﾞﾚｽ
MOVL(498) &14600 D20  ; DB_ST6転送元ｱﾄﾞﾚｽ
MOVL(498) &14700 D22  ; DB_Tmp転送元ｱﾄﾞﾚｽ

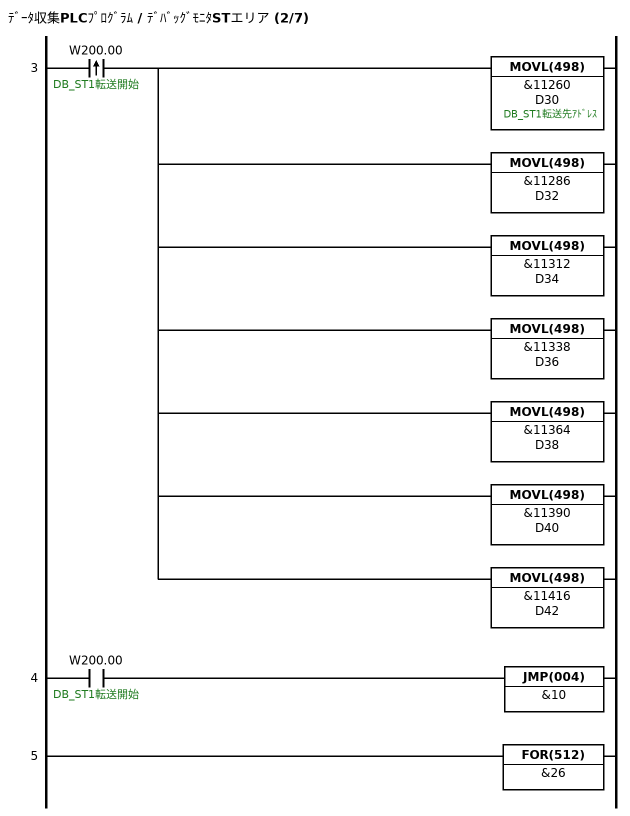
; rung 3
@LD W200.00  ; DB_ST1転送開始
MOVL(498) &11260 D30  ; DB_ST1転送先ｱﾄﾞﾚｽ
MOVL(498) &11286 D32
MOVL(498) &11312 D34
MOVL(498) &11338 D36
MOVL(498) &11364 D38
MOVL(498) &11390 D40
MOVL(498) &11416 D42
; rung 4
LD W200.00  ; DB_ST1転送開始
JMP(004) &10
; rung 5
FOR(512) &26

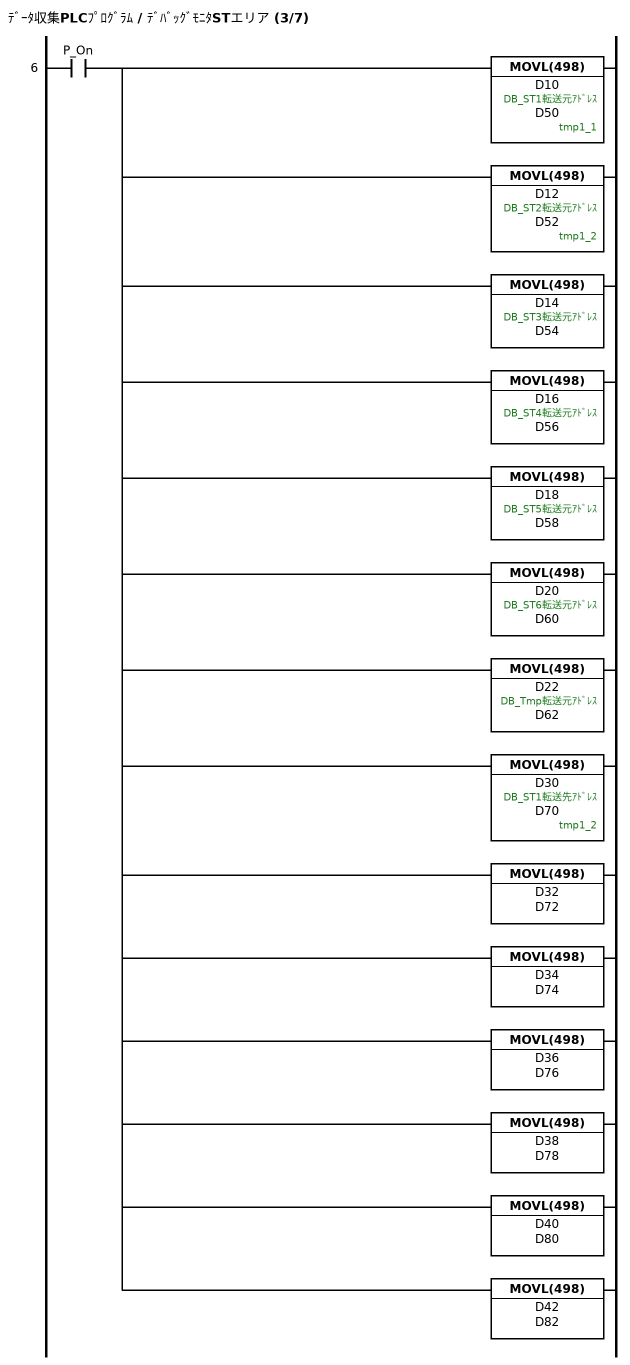
; rung 6
LD P_On
MOVL(498) D10 D50  ; DB_ST1転送元ｱﾄﾞﾚｽ, tmp1_1
MOVL(498) D12 D52  ; DB_ST2転送元ｱﾄﾞﾚｽ, tmp1_2
MOVL(498) D14 D54  ; DB_ST3転送元ｱﾄﾞﾚｽ
MOVL(498) D16 D56  ; DB_ST4転送元ｱﾄﾞﾚｽ
MOVL(498) D18 D58  ; DB_ST5転送元ｱﾄﾞﾚｽ
MOVL(498) D20 D60  ; DB_ST6転送元ｱﾄﾞﾚｽ
MOVL(498) D22 D62  ; DB_Tmp転送元ｱﾄﾞﾚｽ
MOVL(498) D30 D70  ; DB_ST1転送先ｱﾄﾞﾚｽ, tmp1_2
MOVL(498) D32 D72
MOVL(498) D34 D74
MOVL(498) D36 D76
MOVL(498) D38 D78
MOVL(498) D40 D80
MOVL(498) D42 D82

